FUNCTION FC_AlarmExists : BOOL
VAR_INPUT
    SourceName: STRING(255) := '';
	TcSourceInfo	: FB_TcSourceInfo;
	TcEventLogger 	: FB_TcEventLogger;
	TcAlarm	: REFERENCE TO FB_TcAlarm;
	pTcEventEntry	: TcEventEntry;
	EventId	: UDINT;
END_VAR
VAR
	hr	: HRESULT;
END_VAR

TcSourceInfo.sName := CONCAT('PLC.', SourceName);
hr := TcEventLogger.GetAlarm(pTcEventEntry.uuidEventClass, EventId, TcSourceInfo, TcAlarm);

// Create event if not already created
IF NOT SUCCEEDED(hr) THEN		
	hr := TcAlarm.CreateEx(pTcEventEntry, FALSE, TcSourceInfo);
END_IF;	

IF SUCCEEDED(hr) THEN		
	FC_AlarmExists := TRUE;
ELSE
	FC_AlarmExists := FALSE;
END_IF;

END_FUNCTION

(* stored: Version 1.1.0.1, ProductVersion 3.1.4024.15
   POU FC_AlarmExists: Id {bae820b5-4b79-43a8-bf88-2b7d104e2f4e}, SpecialFunc None *)
